FUNCTION WRITE_PROTECTED_DWORD
VAR_INPUT
    Ptr : POINTER TO DWORD;
    Value : DWORD;
END_VAR

Ptr^ := Value;

END_FUNCTION

(* stored: Version 1.1.0.1, ProductVersion 3.1.4022.18
   POU WRITE_PROTECTED_DWORD: Id {adb6e532-53d2-41dc-9582-b0d035315f3a}, SpecialFunc None *)
